{attribute 'qualified_only'}
{attribute 'strict'}
{attribute 'to_string'}
TYPE E_Voltages :
(
	_600V := 600,
	_480V := 480,
	_208V := 208
);
END_TYPE

(* stored: Version 1.1.0.1, ProductVersion 3.1.4026.18
   DUT E_Voltages: Id {2638da28-e565-45bc-91a8-4f063dbefaa7} *)
